TYPE stEMbase :
STRUCT
	sTagName : STRING;
	sDescription : STRING;
END_STRUCT
END_TYPE

(* stored: Version 1.1.0.1, ProductVersion 3.1.4024.12
   DUT stEMbase: Id {8c284a2f-bdb0-40ae-b911-9e30de1f2ace} *)
